PROGRAM MAIN
VAR
END_VAR

END_PROGRAM

(* stored: Version 1.1.0.1
   POU MAIN: Id {6f3d5839-1e33-4585-ad06-48a190c42c62} *)
